PROGRAM IF_RACK_CHECK
VAR_INPUT
	checkIn_A5 : BOOL;
	checkIn_A4 : BOOL;
	checkIn_A3 : BOOL;
	checkIn_A2 : BOOL;
	checkIn_A1 : BOOL;
	checkIn_B5 : BOOL;
	checkIn_B4 : BOOL;
	checkIn_B3 : BOOL;
	checkIn_B2 : BOOL;
	checkIn_B1 : BOOL;
END_VAR
VAR
	infeedRack_A_empty: BOOL;
	infeedRack_B_empty: BOOL;
	turnflag: BOOL;
	turningA: BOOL;
	turningB: BOOL;
	cool_rack_check : UINT;
END_VAR


IF NOT AUTO_MODE.Run_Next_Rack THEN
	RETURN;
END_IF
	
IF COOL_RACK.CR_full THEN
	RETURN;
END_IF

IF INFEED_RACK.FaceA_InWC THEN
	IF INFEED_RACK.A5_Sensor THEN
		checkIn_A5 := TRUE; AUTO_MODE.Run_Next_Rack := FALSE;
	ELSIF INFEED_RACK.A4_Sensor THEN
		checkIn_A4 := TRUE; AUTO_MODE.Run_Next_Rack := FALSE;
	ELSIF INFEED_RACK.A3_Sensor THEN
		checkIn_A3 := TRUE; AUTO_MODE.Run_Next_Rack := FALSE;
	ELSIF INFEED_RACK.A2_Sensor THEN
		checkIn_A2 := TRUE; AUTO_MODE.Run_Next_Rack := FALSE;
	ELSIF INFEED_RACK.A1_Sensor THEN
		checkIn_A1 := TRUE; AUTO_MODE.Run_Next_Rack := FALSE;
	ELSE
		infeedRack_A_empty := TRUE;	
	END_IF
	
ELSIF INFEED_RACK.FaceB_InWC THEN
	IF INFEED_RACK.B5_Sensor THEN
		checkIn_B5 := TRUE; AUTO_MODE.Run_Next_Rack := FALSE;
	ELSIF INFEED_RACK.B4_Sensor THEN
		checkIn_B4 := TRUE; AUTO_MODE.Run_Next_Rack := FALSE;
	ELSIF INFEED_RACK.B3_Sensor THEN
		checkIn_B3 := TRUE; AUTO_MODE.Run_Next_Rack := FALSE;
	ELSIF INFEED_RACK.B2_Sensor THEN
		checkIn_B2 := TRUE; AUTO_MODE.Run_Next_Rack := FALSE;
	ELSIF INFEED_RACK.B1_Sensor THEN
		checkIn_B1 := TRUE; AUTO_MODE.Run_Next_Rack := FALSE;
	ELSE
		infeedRack_B_empty := TRUE;	
	END_IF
END_IF

IF INFEED_RACK.IFRack_Ready and INFEED_RACK.IFRack_TurnReady THEN
	IF infeedRack_A_empty AND NOT turningB THEN
		turningA := TRUE;
		INFEED_RACK.IFRack_arr[1].5 := FALSE; //BtoA
		INFEED_RACK.IFRack_arr[1].4 := TRUE; //AtoB
		INFEED_RACK(bStart_Write:=TRUE);
		IF INFEED_RACK.FaceB_InWC THEN
			turningA := FALSE;
			infeedRack_A_empty := FALSE;
			INFEED_RACK(bStart_Write:=FALSE);
		END_IF
	ELSIF infeedRack_B_empty AND NOT turningA THEN
		turningB := TRUE;
		INFEED_RACK.IFRack_arr[1].4 := FALSE; //AtoB
		INFEED_RACK.IFRack_arr[1].5 := TRUE; //BtoA
		INFEED_RACK(bStart_Write:=TRUE);
		IF INFEED_RACK.FaceA_InWC THEN
			turningB := FALSE;
			infeedRack_B_empty := FALSE;
			INFEED_RACK(bStart_Write:=FALSE);
		END_IF
	END_IF
END_IF

//INFEED_RACK.bStart_Read:=FALSE;
//INFEED_RACK.bStart_Write:=FALSE;

END_PROGRAM

(* stored: Version 1.1.0.1, ProductVersion 3.1.4024.12
   POU IF_RACK_CHECK: Id {4d16c559-2d91-410a-8902-60c712acc471}, SpecialFunc None *)
